{attribute addProperty BoxType "EL6692-0002-0016"}
{attribute addProperty Id "Sync_ModeAT %I*BYTE812TxPDO_toggleAT %I*BOOL819TxPDO_stateAT %I*BOOL817Control_value_update_toggleAT %I*BOOL8114Timestamp_update_toggleAT %I*BOOL8115External_device_not_connectedAT %I*BOOL8116"}
{attribute addProperty CRC "2911881473"}
{attribute addProperty SizeInBites "48"}
{attribute addProperty SizeInBytes "6"}
TYPE SYNC_Inputs_AD8FC901 :
STRUCT
	{attribute addProperty Name "Sync_Mode"}
	Sync_Mode AT %I* : BYTE;
	{attribute addProperty Name "TxPDO_toggle"}
	TxPDO_toggle AT %I* : BOOL;
	{attribute addProperty Name "TxPDO_state"}
	TxPDO_state AT %I* : BOOL;
	{attribute addProperty Name "Control_value_update_toggle"}
	Control_value_update_toggle AT %I* : BOOL;
	{attribute addProperty Name "Timestamp_update_toggle"}
	Timestamp_update_toggle AT %I* : BOOL;
	{attribute addProperty Name "External_device_not_connected"}
	External_device_not_connected AT %I* : BOOL;
END_STRUCT
END_TYPE

(* stored: Version 1.2.0.0, ProductVersion 3.1.4024.9
   DUT SYNC_Inputs_AD8FC901: Id {d4fd7adf-0120-4fbe-bdfc-60afe97842fb} *)
